(* CoDeSys 2.3 export: PUMP_STATION.EXP *)
(* Libraries: ANALYZATION.LIB 5.10.99 09:05:06, IECSFC.LIB 13.4.06 15:51:28, STANDARD.LIB 4.10.05 11:14:46, SYSLIBCALLBACK.LIB 26.10.21 13:46:42, SYSLIBTIME.LIB 26.10.21 13:46:42, SYSTASKINFO.LIB 26.10.21 13:46:42, Util.lib 18.5.10 15:14:28 *)

(* PLC configuration (modules and I/O channels)
PLC110_32 [Root] node -1, in %IB0 out %QB0 {param 1 = PLC110-32_v2; param 2 = 1; param 3 = 1000}
  Fast discrete inputs [I_SIMPLE_INPUT] node 0, in %IB0 out %QB0 {param 1 = Fast discrete inputs; param 2 = 10000}
    AT %IX0.0 [BitInput] Discrete input 1 {param 1 = Enter name}
    AT %IX0.1 [BitInput] Discrete input 2 {param 1 = Enter name}
  Discrete inputs [ID130] node 1, in %IB1 out %QB1 {param 1 = Discrete inputs; param 2 = 16; param 3 = 16}
    discrete_input_first_byte AT %IB1.0 [ByteInput] discrete_input_first_byte {param 1 = Enter name}
    discrete_input_second_byte AT %IB1.1 [ByteInput] discrete input_second_byte {param 1 = Enter name}
  Fast discrete outputs [OWEN_ID570] node 2, in %IB2 out %QB2 {param 1 = Fast discrete outputs; param 2 = FALSE; param 3 = FALSE; param 4 = FALSE; param 5 = FALSE}
    hw_run_id1 AT %QX2.0 [BitOutput] Run hot water invertor drive1 {param 1 = Enter name}
    hw_run_id2 AT %QX2.1 [BitOutput] Run hot water invertor drive2 {param 1 = Enter name}
    ws_run_id1 AT %QX2.2 [BitOutput] Run water supply invertor drive1 {param 1 = Enter name}
    ws_run_id2 AT %QX2.3 [BitOutput] Run water supply invertor drive2 {param 1 = Enter name}
  Discrete outputs [ID131] node 3, in %IB3 out %QB3 {param 1 = Discrete outputs; param 2 = 0; param 3 = 0; param 4 = 0; param 5 = 24}
    AT %QB3.0 [ByteOutput] 8 discrete outputs {param 1 = Enter name}
    AT %QB3.1 [ByteOutput] 8 discrete outputs {param 1 = Enter name}
  Special input [ID103] node 4, in %IB4 out %QB4 {param 1 = Special input}
    AT %IX4.0 [BitInput] Special input {param 1 = Enter name}
  Special output [ID104] node 5, in %IB5 out %QB5 {param 1 = Special output}
    AT %QX5.0 [BitOutput] Special output {param 1 = Enter name}
  ModBus (Master) [MODBUS_MASTER_ID450] node 6, in %IB6 out %QB6 {param 1 = ModBus (Master); param 2 = No}
    AT %QD6.0 [DWordOutput] Last address {param 1 = Enter name}
    AT %QW6.1 [WordOutput] Last error {param 1 = Enter name}
    RS-485-1 [COM1_USART] node 0, in %IB6.0 out %QB6.0 {param 1 = RS-485-1; param 2 = 115200; param 3 = NO PARITY CHECK; param 4 = 8 bits; param 5 = One stop bit; param 6 = RS485; param 7 = RTU; param 8 = 0; param 9 = No}
    Universal Modbus device [ID2000] node 1, in %IB6.1 out %QB6.1 {param 1 = Universal Modbus device; param 2 = 10:0:0:223; param 3 = 150; param 4 = 502; param 5 = Serial; param 6 = 16; param 7 = By poll time; param 8 = 100; param 9 = No; param 10 = 0; param 11 = Trace_mode}
      AT %QB6.1.0 [ComChannel] Command (0xff - Start) {param 1 = Enter name}
      Real input module [ID2007] node 0, in %IB6.1.0 out %QB6.1.0 {param 1 = float input module; param 2 = 4; param 3 = Read holding Registers  (0x03); param 8 = No}
        hw_input_pressure AT %QD6.1.0.0 [FloatOutput] {param 1 = Enter name}
      Register input module [ID2003] node 1, in %IB6.1.1 out %QB6.1.1 {param 1 = Register input module; param 2 = 2; param 3 = Read holding Registers  (0x03); param 8 = No}
        hw_error_input_pressure AT %QW6.1.1.0 [WordOutput] {param 1 = Enter name}
      Real input module [ID2007] node 2, in %IB6.1.2 out %QB6.1.2 {param 1 = float input module; param 2 = 10; param 3 = Read holding Registers  (0x03); param 8 = No}
        hw_output_pressure AT %QD6.1.2.0 [FloatOutput] {param 1 = Enter name}
      Register input module [ID2003] node 3, in %IB6.1.3 out %QB6.1.3 {param 1 = Register input module; param 2 = 8; param 3 = Read holding Registers  (0x03); param 8 = No}
        hw_error_output_pressure AT %QW6.1.3.0 [WordOutput] {param 1 = Enter name}
      Real input module [ID2007] node 4, in %IB6.1.4 out %QB6.1.4 {param 1 = float input module; param 2 = 16; param 3 = Read holding Registers  (0x03); param 8 = No}
        ws_input_pressure AT %QD6.1.4.0 [FloatOutput] {param 1 = Enter name}
      Register input module [ID2003] node 5, in %IB6.1.5 out %QB6.1.5 {param 1 = Register input module; param 2 = 14; param 3 = Read holding Registers  (0x03); param 8 = No}
        ws_error_input_pressure AT %QW6.1.5.0 [WordOutput] {param 1 = Enter name}
      Real input module [ID2007] node 6, in %IB6.1.6 out %QB6.1.6 {param 1 = float input module; param 2 = 22; param 3 = Read holding Registers  (0x03); param 8 = No}
        ws_output_pressure AT %QD6.1.6.0 [FloatOutput] {param 1 = Enter name}
      Register input module [ID2003] node 7, in %IB6.1.7 out %QB6.1.7 {param 1 = Register input module; param 2 = 20; param 3 = Read holding Registers  (0x03); param 8 = No}
        ws_error_output_pressure AT %QW6.1.7.0 [WordOutput] {param 1 = Enter name}
  ModBus (Master) [MODBUS_MASTER_ID450] node 7, in %IB7 out %QB7 {param 1 = ModBus (Master); param 2 = No}
    AT %QD7.0 [DWordOutput] Last address {param 1 = Enter name}
    AT %QW7.1 [WordOutput] Last error {param 1 = Enter name}
    RS-485-1 [COM1_USART] node 0, in %IB7.0 out %QB7.0 {param 1 = RS-485-1; param 2 = 115200; param 3 = NO PARITY CHECK; param 4 = 8 bits; param 5 = One stop bit; param 6 = RS485; param 7 = RTU; param 8 = 0; param 9 = No}
    Universal Modbus device [ID2000] node 1, in %IB7.1 out %QB7.1 {param 1 = Universal Modbus device; param 2 = 10:0:0:223; param 3 = 150; param 4 = 502; param 5 = Serial; param 6 = 32; param 7 = By poll time; param 8 = 100; param 9 = No; param 10 = 0; param 11 = Trace_mode}
      AT %QB7.1.0 [ComChannel] Command (0xff - Start) {param 1 = Enter name}
      Register output module [ID2004] node 0, in %IB7.1.0 out %QB7.1.0 {param 1 = Register; param 2 = 0; param 3 = Write multiple registers(0x10); param 8 = No}
        hw_output_value_id1 AT %QW7.1.0.0 [WordOutput] {param 1 = Enter name}
      Register output module [ID2004] node 1, in %IB7.1.1 out %QB7.1.1 {param 1 = Register; param 2 = 1; param 3 = Write multiple registers(0x10); param 8 = No}
        hw_output_value_id2 AT %QW7.1.1.0 [WordOutput] {param 1 = Enter name}
      Register output module [ID2004] node 2, in %IB7.1.2 out %QB7.1.2 {param 1 = Register; param 2 = 2; param 3 = Write multiple registers(0x10); param 8 = No}
        ws_output_value_id1 AT %QW7.1.2.0 [WordOutput] {param 1 = Enter name}
      Register output module [ID2004] node 3, in %IB7.1.3 out %QB7.1.3 {param 1 = Register; param 2 = 3; param 3 = Write multiple registers(0x10); param 8 = No}
        ws_output_value_id2 AT %QW7.1.3.0 [WordOutput] {param 1 = Enter name}
      Register output module [ID2004] node 4, in %IB7.1.4 out %QB7.1.4 {param 1 = Register; param 2 = 4; param 3 = Write multiple registers(0x10); param 8 = No}
        AT %QW7.1.4.0 [WordOutput] {param 1 = Enter name}
      Register output module [ID2004] node 5, in %IB7.1.5 out %QB7.1.5 {param 1 = Register; param 2 = 5; param 3 = Write multiple registers(0x10); param 8 = No}
        AT %QW7.1.5.0 [WordOutput] {param 1 = Enter name}
      Register output module [ID2004] node 6, in %IB7.1.6 out %QB7.1.6 {param 1 = Register; param 2 = 6; param 3 = Write multiple registers(0x10); param 8 = No}
        AT %QW7.1.6.0 [WordOutput] {param 1 = Enter name}
      Register output module [ID2004] node 7, in %IB7.1.7 out %QB7.1.7 {param 1 = Register; param 2 = 7; param 3 = Write multiple registers(0x10); param 8 = No}
        AT %QW7.1.7.0 [WordOutput] {param 1 = Enter name}
  ModBus (slave) [MODBUS_ID400] node 8, in %IB8 out %QB8 {param 1 = ModBus (slave); param 2 = 1}
    Modbus [MODBUS_ID302] node 0, in %IB8.0 out %QB8.0 {param 1 = Modbus}
      RS-232 [COM2_USART] node 0, in %IB8.0.0 out %QB8.0.0 {param 1 = RS-232; param 2 = 115200; param 3 = NO PARITY CHECK; param 4 = 8 bits; param 5 = One stop bit; param 6 = RS232; param 7 = RTU; param 8 = 0; param 9 = No}
    8 bits [8Bit] node 1, in %IB8.1 out %QB8.1 {param 1 = 8 bit}
      AT %QB8.1.0 [ByteOutput] {param 1 = Enter name}
    8 bits [8Bit] node 2, in %IB8.2 out %QB8.2 {param 1 = 8 bit}
      AT %QB8.2.0 [ByteOutput] {param 1 = Enter name}
    8 bits [8Bit] node 3, in %IB8.3 out %QB8.3 {param 1 = 8 bit}
      AT %QB8.3.0 [ByteOutput] {param 1 = Enter name}
    8 bits [8Bit] node 4, in %IB8.4 out %QB8.4 {param 1 = 8 bit}
      AT %QB8.4.0 [ByteOutput] {param 1 = Enter name}
    2 byte [Register] node 5, in %IB8.5 out %QB8.5 {param 1 = 2 byte}
      hw_pivot_single AT %QW8.5.0 [WordOutput] {param 1 = Enter name}
    2 byte [Register] node 6, in %IB8.6 out %QB8.6 {param 1 = 2 byte}
      hw_pivot_cascade AT %QW8.6.0 [WordOutput] {param 1 = Enter name}
    2 byte [Register] node 7, in %IB8.7 out %QB8.7 {param 1 = 2 byte}
      hw_cycle_set_hours AT %QW8.7.0 [WordOutput] {param 1 = Enter name}
    2 byte [Register] node 8, in %IB8.8 out %QB8.8 {param 1 = 2 byte}
      hw_cycle_set_minutes AT %QW8.8.0 [WordOutput] {param 1 = Enter name}
    2 byte [Register] node 9, in %IB8.9 out %QB8.9 {param 1 = 2 byte}
      hw_cycle_set_seconds AT %QW8.9.0 [WordOutput] {param 1 = Enter name}
    2 byte [Register] node 10, in %IB8.10 out %QB8.10 {param 1 = 2 byte}
      hw_cascade_delay_on_hours AT %QW8.10.0 [WordOutput] {param 1 = Enter name}
    2 byte [Register] node 11, in %IB8.11 out %QB8.11 {param 1 = 2 byte}
      hw_cascade_delay_on_minutes AT %QW8.11.0 [WordOutput] {param 1 = Enter name}
    2 byte [Register] node 12, in %IB8.12 out %QB8.12 {param 1 = 2 byte}
      hw_cascade_delay_on_seconds AT %QW8.12.0 [WordOutput] {param 1 = Enter name}
    2 byte [Register] node 13, in %IB8.13 out %QB8.13 {param 1 = 2 byte}
      hw_cascade_delay_off_hours AT %QW8.13.0 [WordOutput] {param 1 = Enter name}
    2 byte [Register] node 14, in %IB8.14 out %QB8.14 {param 1 = 2 byte}
      hw_cascade_delay_off_minutes AT %QW8.14.0 [WordOutput] {param 1 = Enter name}
    2 byte [Register] node 15, in %IB8.15 out %QB8.15 {param 1 = 2 byte}
      hw_cascade_delay_off_seconds AT %QW8.15.0 [WordOutput] {param 1 = Enter name}
    2 byte [Register] node 16, in %IB8.16 out %QB8.16 {param 1 = 2 byte}
      ws_pivot_single AT %QW8.16.0 [WordOutput] {param 1 = Enter name}
    2 byte [Register] node 17, in %IB8.17 out %QB8.17 {param 1 = 2 byte}
      ws_pivot_cascade AT %QW8.17.0 [WordOutput] {param 1 = Enter name}
    2 byte [Register] node 18, in %IB8.18 out %QB8.18 {param 1 = 2 byte}
      ws_cycle_set_hours AT %QW8.18.0 [WordOutput] {param 1 = Enter name}
    2 byte [Register] node 19, in %IB8.19 out %QB8.19 {param 1 = 2 byte}
      ws_cycle_set_minutes AT %QW8.19.0 [WordOutput] {param 1 = Enter name}
    2 byte [Register] node 20, in %IB8.20 out %QB8.20 {param 1 = 2 byte}
      ws_cycle_set_seconds AT %QW8.20.0 [WordOutput] {param 1 = Enter name}
    2 byte [Register] node 21, in %IB8.21 out %QB8.21 {param 1 = 2 byte}
      ws_cascade_delay_on_hours AT %QW8.21.0 [WordOutput] {param 1 = Enter name}
    2 byte [Register] node 22, in %IB8.22 out %QB8.22 {param 1 = 2 byte}
      ws_cascade_delay_on_minutes AT %QW8.22.0 [WordOutput] {param 1 = Enter name}
    2 byte [Register] node 23, in %IB8.23 out %QB8.23 {param 1 = 2 byte}
      ws_cascade_delay_on_seconds AT %QW8.23.0 [WordOutput] {param 1 = Enter name}
    2 byte [Register] node 24, in %IB8.24 out %QB8.24 {param 1 = 2 byte}
      ws_cascade_delay_off_hours AT %QW8.24.0 [WordOutput] {param 1 = Enter name}
    2 byte [Register] node 25, in %IB8.25 out %QB8.25 {param 1 = 2 byte}
      ws_cascade_delay_off_minutes AT %QW8.25.0 [WordOutput] {param 1 = Enter name}
    2 byte [Register] node 26, in %IB8.26 out %QB8.26 {param 1 = 2 byte}
      ws_cascade_delay_off_seconds AT %QW8.26.0 [WordOutput] {param 1 = Enter name}
    Float [Float] node 27, in %IB8.27 out %QB8.27 {param 1 = float}
      hw_set_point_pressure AT %QD8.27.0 [FloatOutput] {param 1 = Enter name}
    Float [Float] node 28, in %IB8.28 out %QB8.28 {param 1 = float}
      ws_set_point_pressure AT %QD8.28.0 [FloatOutput] {param 1 = Enter name}
    Float [Float] node 29, in %IB8.29 out %QB8.29 {param 1 = float}
      hw_min_measure_range_input AT %QD8.29.0 [FloatOutput] {param 1 = Enter name}
    Float [Float] node 30, in %IB8.30 out %QB8.30 {param 1 = float}
      hw_max_measure_range_input AT %QD8.30.0 [FloatOutput] {param 1 = Enter name}
    Float [Float] node 31, in %IB8.31 out %QB8.31 {param 1 = float}
      hw_min_measure_range_output AT %QD8.31.0 [FloatOutput] {param 1 = Enter name}
    Float [Float] node 32, in %IB8.32 out %QB8.32 {param 1 = float}
      hw_max_measure_range_output AT %QD8.32.0 [FloatOutput] {param 1 = Enter name}
    Float [Float] node 33, in %IB8.33 out %QB8.33 {param 1 = float}
      ws_min_measure_range_input AT %QD8.33.0 [FloatOutput] {param 1 = Enter name}
    Float [Float] node 34, in %IB8.34 out %QB8.34 {param 1 = float}
      ws_max_measure_range_input AT %QD8.34.0 [FloatOutput] {param 1 = Enter name}
    Float [Float] node 35, in %IB8.35 out %QB8.35 {param 1 = float}
      ws_min_measure_range_output AT %QD8.35.0 [FloatOutput] {param 1 = Enter name}
    Float [Float] node 36, in %IB8.36 out %QB8.36 {param 1 = float}
      ws_max_measure_range_output AT %QD8.36.0 [FloatOutput] {param 1 = Enter name}
    Float [Float] node 37, in %IB8.37 out %QB8.37 {param 1 = float}
      hw_input_pressure_bar AT %QD8.37.0 [FloatOutput] {param 1 = Enter name}
    Float [Float] node 38, in %IB8.38 out %QB8.38 {param 1 = float}
      hw_output_pressure_bar AT %QD8.38.0 [FloatOutput] {param 1 = Enter name}
    Float [Float] node 39, in %IB8.39 out %QB8.39 {param 1 = float}
      ws_input_pressure_bar AT %QD8.39.0 [FloatOutput] {param 1 = Enter name}
    Float [Float] node 40, in %IB8.40 out %QB8.40 {param 1 = float}
      ws_output_pressure_bar AT %QD8.40.0 [FloatOutput] {param 1 = Enter name}
    Float [Float] node 41, in %IB8.41 out %QB8.41 {param 1 = float}
      hw_frequency_id1 AT %QD8.41.0 [FloatOutput] {param 1 = Enter name}
    Float [Float] node 42, in %IB8.42 out %QB8.42 {param 1 = float}
      hw_frequency_id2 AT %QD8.42.0 [FloatOutput] {param 1 = Enter name}
    Float [Float] node 43, in %IB8.43 out %QB8.43 {param 1 = float}
      ws_frequency_id1 AT %QD8.43.0 [FloatOutput] {param 1 = Enter name}
    Float [Float] node 44, in %IB8.44 out %QB8.44 {param 1 = float}
      ws_frequency_id2 AT %QD8.44.0 [FloatOutput] {param 1 = Enter name}
    2 byte [Register] node 45, in %IB8.45 out %QB8.45 {param 1 = 2 byte}
      hw_alarm_error_code AT %QW8.45.0 [WordOutput] {param 1 = Enter name}
    2 byte [Register] node 46, in %IB8.46 out %QB8.46 {param 1 = 2 byte}
      ws_alarm_error_code AT %QW8.46.0 [WordOutput] {param 1 = Enter name}
    Float [Float] node 47, in %IB8.47 out %QB8.47 {param 1 = float}
      hw_manual_set_frequency_id1 AT %QD8.47.0 [FloatOutput] {param 1 = Enter name}
    Float [Float] node 48, in %IB8.48 out %QB8.48 {param 1 = float}
      hw_manual_set_frequency_id2 AT %QD8.48.0 [FloatOutput] {param 1 = Enter name}
    Float [Float] node 49, in %IB8.49 out %QB8.49 {param 1 = float}
      ws_manual_set_frequency_id1 AT %QD8.49.0 [FloatOutput] {param 1 = Enter name}
    Float [Float] node 50, in %IB8.50 out %QB8.50 {param 1 = float}
      ws_manual_set_frequency_id2 AT %QD8.50.0 [FloatOutput] {param 1 = Enter name}
    2 byte [Register] node 51, in %IB8.51 out %QB8.51 {param 1 = 2 byte}
      AT %QW8.51.0 [WordOutput] {param 1 = Enter name}
    2 byte [Register] node 52, in %IB8.52 out %QB8.52 {param 1 = 2 byte}
      AT %QW8.52.0 [WordOutput] {param 1 = Enter name}
    2 byte [Register] node 53, in %IB8.53 out %QB8.53 {param 1 = 2 byte}
      AT %QW8.53.0 [WordOutput] {param 1 = Enter name}
    2 byte [Register] node 54, in %IB8.54 out %QB8.54 {param 1 = 2 byte}
      AT %QW8.54.0 [WordOutput] {param 1 = Enter name}
    2 byte [Register] node 55, in %IB8.55 out %QB8.55 {param 1 = 2 byte}
      AT %QW8.55.0 [WordOutput] {param 1 = Enter name}
    2 byte [Register] node 56, in %IB8.56 out %QB8.56 {param 1 = 2 byte}
      AT %QW8.56.0 [WordOutput] {param 1 = Enter name}
    2 byte [Register] node 57, in %IB8.57 out %QB8.57 {param 1 = 2 byte}
      AT %QW8.57.0 [WordOutput] {param 1 = Enter name}
    2 byte [Register] node 58, in %IB8.58 out %QB8.58 {param 1 = 2 byte}
      AT %QW8.58.0 [WordOutput] {param 1 = Enter name}
    2 byte [Register] node 59, in %IB8.59 out %QB8.59 {param 1 = 2 byte}
      AT %QW8.59.0 [WordOutput] {param 1 = Enter name}
    2 byte [Register] node 60, in %IB8.60 out %QB8.60 {param 1 = 2 byte}
      AT %QW8.60.0 [WordOutput] {param 1 = Enter name}
    2 byte [Register] node 61, in %IB8.61 out %QB8.61 {param 1 = 2 byte}
      AT %QW8.61.0 [WordOutput] {param 1 = Enter name}
    2 byte [Register] node 62, in %IB8.62 out %QB8.62 {param 1 = 2 byte}
      AT %QW8.62.0 [WordOutput] {param 1 = Enter name}
    2 byte [Register] node 63, in %IB8.63 out %QB8.63 {param 1 = 2 byte}
      AT %QW8.63.0 [WordOutput] {param 1 = Enter name}
    2 byte [Register] node 64, in %IB8.64 out %QB8.64 {param 1 = 2 byte}
      AT %QW8.64.0 [WordOutput] {param 1 = Enter name}
    2 byte [Register] node 65, in %IB8.65 out %QB8.65 {param 1 = 2 byte}
      AT %QW8.65.0 [WordOutput] {param 1 = Enter name}
    2 byte [Register] node 66, in %IB8.66 out %QB8.66 {param 1 = 2 byte}
      AT %QW8.66.0 [WordOutput] {param 1 = Enter name}
    2 byte [Register] node 67, in %IB8.67 out %QB8.67 {param 1 = 2 byte}
      AT %QW8.67.0 [WordOutput] {param 1 = Enter name}
    2 byte [Register] node 68, in %IB8.68 out %QB8.68 {param 1 = 2 byte}
      AT %QW8.68.0 [WordOutput] {param 1 = Enter name}
    2 byte [Register] node 69, in %IB8.69 out %QB8.69 {param 1 = 2 byte}
      AT %QW8.69.0 [WordOutput] {param 1 = Enter name}
    2 byte [Register] node 70, in %IB8.70 out %QB8.70 {param 1 = 2 byte}
      AT %QW8.70.0 [WordOutput] {param 1 = Enter name}
    2 byte [Register] node 71, in %IB8.71 out %QB8.71 {param 1 = 2 byte}
      AT %QW8.71.0 [WordOutput] {param 1 = Enter name}
    2 byte [Register] node 72, in %IB8.72 out %QB8.72 {param 1 = 2 byte}
      AT %QW8.72.0 [WordOutput] {param 1 = Enter name}
    2 byte [Register] node 73, in %IB8.73 out %QB8.73 {param 1 = 2 byte}
      AT %QW8.73.0 [WordOutput] {param 1 = Enter name}
    2 byte [Register] node 74, in %IB8.74 out %QB8.74 {param 1 = 2 byte}
      AT %QW8.74.0 [WordOutput] {param 1 = Enter name}
    2 byte [Register] node 75, in %IB8.75 out %QB8.75 {param 1 = 2 byte}
      AT %QW8.75.0 [WordOutput] {param 1 = Enter name}
    2 byte [Register] node 76, in %IB8.76 out %QB8.76 {param 1 = 2 byte}
      AT %QW8.76.0 [WordOutput] {param 1 = Enter name}
    2 byte [Register] node 77, in %IB8.77 out %QB8.77 {param 1 = 2 byte}
      AT %QW8.77.0 [WordOutput] {param 1 = Enter name}
    2 byte [Register] node 78, in %IB8.78 out %QB8.78 {param 1 = 2 byte}
      AT %QW8.78.0 [WordOutput] {param 1 = Enter name}
    2 byte [Register] node 79, in %IB8.79 out %QB8.79 {param 1 = 2 byte}
      AT %QW8.79.0 [WordOutput] {param 1 = Enter name}
    2 byte [Register] node 80, in %IB8.80 out %QB8.80 {param 1 = 2 byte}
      AT %QW8.80.0 [WordOutput] {param 1 = Enter name}
    2 byte [Register] node 81, in %IB8.81 out %QB8.81 {param 1 = 2 byte}
      AT %QW8.81.0 [WordOutput] {param 1 = Enter name}
    2 byte [Register] node 82, in %IB8.82 out %QB8.82 {param 1 = 2 byte}
      AT %QW8.82.0 [WordOutput] {param 1 = Enter name}
    2 byte [Register] node 83, in %IB8.83 out %QB8.83 {param 1 = 2 byte}
      AT %QW8.83.0 [WordOutput] {param 1 = Enter name}
    2 byte [Register] node 84, in %IB8.84 out %QB8.84 {param 1 = 2 byte}
      AT %QW8.84.0 [WordOutput] {param 1 = Enter name}
    2 byte [Register] node 85, in %IB8.85 out %QB8.85 {param 1 = 2 byte}
      AT %QW8.85.0 [WordOutput] {param 1 = Enter name}
    2 byte [Register] node 86, in %IB8.86 out %QB8.86 {param 1 = 2 byte}
      AT %QW8.86.0 [WordOutput] {param 1 = Enter name}
    2 byte [Register] node 87, in %IB8.87 out %QB8.87 {param 1 = 2 byte}
      AT %QW8.87.0 [WordOutput] {param 1 = Enter name}
    2 byte [Register] node 88, in %IB8.88 out %QB8.88 {param 1 = 2 byte}
      AT %QW8.88.0 [WordOutput] {param 1 = Enter name}
    2 byte [Register] node 89, in %IB8.89 out %QB8.89 {param 1 = 2 byte}
      AT %QW8.89.0 [WordOutput] {param 1 = Enter name}
    2 byte [Register] node 90, in %IB8.90 out %QB8.90 {param 1 = 2 byte}
      AT %QW8.90.0 [WordOutput] {param 1 = Enter name}
    2 byte [Register] node 91, in %IB8.91 out %QB8.91 {param 1 = 2 byte}
      AT %QW8.91.0 [WordOutput] {param 1 = Enter name}
    2 byte [Register] node 92, in %IB8.92 out %QB8.92 {param 1 = 2 byte}
      AT %QW8.92.0 [WordOutput] {param 1 = Enter name}
    2 byte [Register] node 93, in %IB8.93 out %QB8.93 {param 1 = 2 byte}
      AT %QW8.93.0 [WordOutput] {param 1 = Enter name}
    2 byte [Register] node 94, in %IB8.94 out %QB8.94 {param 1 = 2 byte}
      AT %QW8.94.0 [WordOutput] {param 1 = Enter name}
    2 byte [Register] node 95, in %IB8.95 out %QB8.95 {param 1 = 2 byte}
      AT %QW8.95.0 [WordOutput] {param 1 = Enter name}
    2 byte [Register] node 96, in %IB8.96 out %QB8.96 {param 1 = 2 byte}
      AT %QW8.96.0 [WordOutput] {param 1 = Enter name}
    2 byte [Register] node 97, in %IB8.97 out %QB8.97 {param 1 = 2 byte}
      AT %QW8.97.0 [WordOutput] {param 1 = Enter name}
    2 byte [Register] node 98, in %IB8.98 out %QB8.98 {param 1 = 2 byte}
      AT %QW8.98.0 [WordOutput] {param 1 = Enter name}
    2 byte [Register] node 99, in %IB8.99 out %QB8.99 {param 1 = 2 byte}
      AT %QW8.99.0 [WordOutput] {param 1 = Enter name}
    2 byte [Register] node 100, in %IB8.100 out %QB8.100 {param 1 = 2 byte}
      AT %QW8.100.0 [WordOutput] {param 1 = Enter name}
    2 byte [Register] node 101, in %IB8.101 out %QB8.101 {param 1 = 2 byte}
      AT %QW8.101.0 [WordOutput] {param 1 = Enter name}
    2 byte [Register] node 102, in %IB8.102 out %QB8.102 {param 1 = 2 byte}
      AT %QW8.102.0 [WordOutput] {param 1 = Enter name}
    2 byte [Register] node 103, in %IB8.103 out %QB8.103 {param 1 = 2 byte}
      AT %QW8.103.0 [WordOutput] {param 1 = Enter name}
    2 byte [Register] node 104, in %IB8.104 out %QB8.104 {param 1 = 2 byte}
      AT %QW8.104.0 [WordOutput] {param 1 = Enter name}
    2 byte [Register] node 105, in %IB8.105 out %QB8.105 {param 1 = 2 byte}
      AT %QW8.105.0 [WordOutput] {param 1 = Enter name}
    2 byte [Register] node 106, in %IB8.106 out %QB8.106 {param 1 = 2 byte}
      AT %QW8.106.0 [WordOutput] {param 1 = Enter name}
    2 byte [Register] node 107, in %IB8.107 out %QB8.107 {param 1 = 2 byte}
      AT %QW8.107.0 [WordOutput] {param 1 = Enter name}
    2 byte [Register] node 108, in %IB8.108 out %QB8.108 {param 1 = 2 byte}
      AT %QW8.108.0 [WordOutput] {param 1 = Enter name}
    2 byte [Register] node 109, in %IB8.109 out %QB8.109 {param 1 = 2 byte}
      AT %QW8.109.0 [WordOutput] {param 1 = Enter name}
    2 byte [Register] node 110, in %IB8.110 out %QB8.110 {param 1 = 2 byte}
      AT %QW8.110.0 [WordOutput] {param 1 = Enter name}
    2 byte [Register] node 111, in %IB8.111 out %QB8.111 {param 1 = 2 byte}
      AT %QW8.111.0 [WordOutput] {param 1 = Enter name}
    2 byte [Register] node 112, in %IB8.112 out %QB8.112 {param 1 = 2 byte}
      AT %QW8.112.0 [WordOutput] {param 1 = Enter name}
    2 byte [Register] node 113, in %IB8.113 out %QB8.113 {param 1 = 2 byte}
      AT %QW8.113.0 [WordOutput] {param 1 = Enter name}
    2 byte [Register] node 114, in %IB8.114 out %QB8.114 {param 1 = 2 byte}
      AT %QW8.114.0 [WordOutput] {param 1 = Enter name}
    2 byte [Register] node 115, in %IB8.115 out %QB8.115 {param 1 = 2 byte}
      AT %QW8.115.0 [WordOutput] {param 1 = Enter name}
    2 byte [Register] node 116, in %IB8.116 out %QB8.116 {param 1 = 2 byte}
      AT %QW8.116.0 [WordOutput] {param 1 = Enter name}
    2 byte [Register] node 117, in %IB8.117 out %QB8.117 {param 1 = 2 byte}
      AT %QW8.117.0 [WordOutput] {param 1 = Enter name}
    2 byte [Register] node 118, in %IB8.118 out %QB8.118 {param 1 = 2 byte}
      AT %QW8.118.0 [WordOutput] {param 1 = Enter name}
    2 byte [Register] node 119, in %IB8.119 out %QB8.119 {param 1 = 2 byte}
      AT %QW8.119.0 [WordOutput] {param 1 = Enter name}
    2 byte [Register] node 120, in %IB8.120 out %QB8.120 {param 1 = 2 byte}
      AT %QW8.120.0 [WordOutput] {param 1 = Enter name}
    2 byte [Register] node 121, in %IB8.121 out %QB8.121 {param 1 = 2 byte}
      AT %QW8.121.0 [WordOutput] {param 1 = Enter name}
    2 byte [Register] node 122, in %IB8.122 out %QB8.122 {param 1 = 2 byte}
      AT %QW8.122.0 [WordOutput] {param 1 = Enter name}
    2 byte [Register] node 123, in %IB8.123 out %QB8.123 {param 1 = 2 byte}
      AT %QW8.123.0 [WordOutput] {param 1 = Enter name}
    2 byte [Register] node 124, in %IB8.124 out %QB8.124 {param 1 = 2 byte}
      AT %QW8.124.0 [WordOutput] {param 1 = Enter name}
    2 byte [Register] node 125, in %IB8.125 out %QB8.125 {param 1 = 2 byte}
      AT %QW8.125.0 [WordOutput] {param 1 = Enter name}
    2 byte [Register] node 126, in %IB8.126 out %QB8.126 {param 1 = 2 byte}
      AT %QW8.126.0 [WordOutput] {param 1 = Enter name}
    2 byte [Register] node 127, in %IB8.127 out %QB8.127 {param 1 = 2 byte}
      AT %QW8.127.0 [WordOutput] {param 1 = Enter name}
    2 byte [Register] node 128, in %IB8.128 out %QB8.128 {param 1 = 2 byte}
      AT %QW8.128.0 [WordOutput] {param 1 = Enter name}
    2 byte [Register] node 129, in %IB8.129 out %QB8.129 {param 1 = 2 byte}
      AT %QW8.129.0 [WordOutput] {param 1 = Enter name}
    2 byte [Register] node 130, in %IB8.130 out %QB8.130 {param 1 = 2 byte}
      AT %QW8.130.0 [WordOutput] {param 1 = Enter name}
    2 byte [Register] node 131, in %IB8.131 out %QB8.131 {param 1 = 2 byte}
      AT %QW8.131.0 [WordOutput] {param 1 = Enter name}
*)

(* Data type in CascadeMode *)
TYPE classInfoCascade :

STRUCT
	pivot:INT;
	error_message:STRING(79);
	error_code: WORD;
	cascade_pump1:classInfoCascadePump;
	cascade_pump2:classInfoCascadePump;
	cascade_pump3:classInfoCascadePump;
	cascade_pump4:classInfoCascadePump;
	cascade_pump5:classInfoCascadePump;
	cascade_pump6:classInfoCascadePump;
	cascade_pump7:classInfoCascadePump;
	cascade_pump8:classInfoCascadePump;
END_STRUCT

END_TYPE

(* Data type in CascadeMode *)
TYPE classInfoCascadePump :

STRUCT
	cascade_pump:BOOL := FALSE;  (*ï¿½ï¿½ï¿½ï¿½ï¿½ï¿½ ï¿½ï¿½ï¿½ï¿½ï¿½ï¿½ ï¿½ï¿½ï¿½ï¿½ï¿½ï¿½*)
	manual:INT := 40;  (*Hz*)
END_STRUCT

END_TYPE

(* Data type in CycleMode *)
TYPE classInfoCycle :

STRUCT
	run_timer: BOOL; (* status work *)
	working_time: TIME; (* pump working time  *)
	pump_number: INT;  (* number working pump *)
	error_code:  WORD;
END_STRUCT

END_TYPE

(* Data type in InvertorDrive/set_auto_invertor_drive *)
TYPE classSetAutoInvertorDrive :

STRUCT
	auto:BOOL := FALSE;
	direct_logic:BOOL := TRUE;  (* ï¿½ï¿½ï¿½ï¿½ ï¿½ï¿½ï¿½ï¿½ï¿½ï¿½ï¿½/ï¿½ï¿½ï¿½ï¿½ï¿½ï¿½ï¿½ï¿½ï¿½ ï¿½ï¿½ï¿½ï¿½ï¿½ï¿½ï¿½ï¿½ï¿½ï¿½; ï¿½ï¿½ï¿½ ï¿½ï¿½ï¿½ï¿½ï¿½ï¿½ï¿½ï¿½ ï¿½ï¿½ï¿½ï¿½ï¿½ï¿½ï¿½ï¿½ï¿½ï¿½ ï¿½ï¿½ï¿½ï¿½ ï¿½ï¿½ï¿½ï¿½ï¿½ï¿½ï¿½ï¿½ ï¿½ï¿½ï¿½ï¿½ï¿½ï¿½ï¿½ï¿½ï¿½ï¿½ï¿½ï¿½ï¿½ï¿½ ï¿½ï¿½ï¿½ï¿½ï¿½ï¿½ï¿½ï¿½ ï¿½ï¿½ï¿½ï¿½ ï¿½ï¿½ï¿½ï¿½ï¿½ï¿½ï¿½, ï¿½ï¿½ï¿½ï¿½ï¿½ï¿½ï¿½ï¿½ ï¿½ï¿½ï¿½ï¿½ï¿½ï¿½ï¿½ ï¿½ï¿½ï¿½ï¿½ï¿½ï¿½ï¿½ï¿½ï¿½ï¿½ï¿½, ï¿½ ï¿½ï¿½ï¿½ï¿½ï¿½ï¿½ï¿½ï¿½*)
	set_point:REAL := 0;  (* ï¿½ï¿½ï¿½ï¿½ï¿½ï¿½ï¿½, ï¿½ï¿½ï¿½ï¿½ï¿½ï¿½ï¿½ï¿½ ï¿½ ï¿½ï¿½ï¿½ï¿½ï¿½ï¿½ï¿½ï¿½ ï¿½ï¿½ï¿½ï¿½ï¿½ï¿½ï¿½ï¿½ï¿½ ï¿½ï¿½ï¿½ï¿½ï¿½ï¿½ï¿½ï¿½ï¿½ï¿½ï¿½ï¿½ï¿½ï¿½ ï¿½ï¿½ï¿½ï¿½ï¿½ï¿½ï¿½ï¿½ *)
	value:REAL := 0;  (* ï¿½ï¿½ï¿½ï¿½ï¿½ï¿½ï¿½ ï¿½ï¿½ï¿½ï¿½ï¿½ï¿½ï¿½ï¿½ ï¿½ï¿½ï¿½ï¿½ï¿½ï¿½ï¿½ï¿½ï¿½ï¿½ï¿½ï¿½ï¿½ï¿½ ï¿½ï¿½ï¿½ï¿½ï¿½ï¿½ï¿½ï¿½, ï¿½ï¿½ï¿½ï¿½ï¿½ï¿½ï¿½ï¿½ï¿½ï¿½ ï¿½ ï¿½ï¿½ï¿½ï¿½ï¿½ï¿½ï¿½ *)
	P:REAL := 2;  (* ï¿½ï¿½ï¿½ï¿½ï¿½ï¿½ï¿½ï¿½ï¿½ï¿½ï¿½ï¿½ï¿½ï¿½ï¿½ï¿½ ï¿½ï¿½ï¿½ï¿½ï¿½ï¿½ï¿½ï¿½ï¿½ï¿½ï¿½ ï¿½ï¿½ï¿½ï¿½ï¿½ï¿½ï¿½ï¿½ï¿½ï¿½, ï¿½ï¿½ï¿½ ï¿½ï¿½ï¿½ï¿½ï¿½ï¿½ï¿½ï¿½ï¿½ï¿½ ï¿½ï¿½ï¿½ï¿½ï¿½ ï¿½ï¿½ï¿½ï¿½ï¿½ï¿½ï¿½ï¿½ï¿½ï¿½ ï¿½ï¿½ï¿½ï¿½ï¿½ï¿½ï¿½ï¿½ï¿½ï¿½ ï¿½ï¿½ï¿½ï¿½ï¿½ï¿½ï¿½*)
	I:INT := 10;  (* ï¿½ï¿½ï¿½ï¿½ï¿½ï¿½ï¿½ï¿½ï¿½ï¿½ï¿½ï¿½ ï¿½ï¿½ï¿½ï¿½ï¿½ï¿½ï¿½ï¿½ï¿½ï¿½ï¿½ ï¿½ï¿½ï¿½ï¿½ï¿½ï¿½ï¿½ï¿½ï¿½ï¿½, ï¿½ï¿½ï¿½ï¿½ï¿½ ï¿½ ï¿½ï¿½ï¿½ï¿½ï¿½ï¿½ï¿½ï¿½ *)
	D:INT := 0;  (* ï¿½ï¿½ï¿½ï¿½ï¿½ï¿½ï¿½ï¿½ï¿½ï¿½ï¿½ï¿½ï¿½ï¿½ï¿½ï¿½ ï¿½ï¿½ï¿½ï¿½ï¿½ï¿½ï¿½ï¿½ï¿½ï¿½ï¿½ ï¿½ï¿½ï¿½ï¿½ï¿½ï¿½ï¿½ï¿½ï¿½ï¿½, ï¿½ï¿½ï¿½ï¿½ï¿½ ï¿½ ï¿½ï¿½ï¿½ï¿½ï¿½ï¿½ï¿½ï¿½ *)
END_STRUCT

END_TYPE

(* Data type in InvertorDrive/set_limit_frequency *)
TYPE classSetLimitFrequency :

STRUCT
	manual:REAL;  (* Hz *)
	min_range:REAL;  (* Hz *)
	max_range:REAL;  (* Hz *)
END_STRUCT

END_TYPE

(* Data type in InvertorDrive *)
TYPE classAlarmInvertorDrive :

STRUCT
	external_alarm:STRING(79);
	fault_invertor_drive:STRING(79);
END_STRUCT

END_TYPE

(* Data type in InvertorDrive *)
TYPE classInfoInvertorDrive :

STRUCT
	active:BOOL;
	status_run:STRING(79);
	set_pid:classSetPid;
	alarm:classAlarmInvertorDrive;
	frequency:REAL;  (* Hz *)
	aout_frequency:REAL;  (* mA *)
	run:BOOL;
	reset_fault:BOOL;
END_STRUCT

END_TYPE

(* Data type in InvertorDrive *)
TYPE classInvertorDrive :

STRUCT
	discrete_inputs:classInvertorDriveDiscreteInputs;
	discrete_outputs:classInvertorDriveDiscreteOutputs;
	analog_input:classInvertorDriveAnalogInputs;
	analog_output:classInvertorDriveAnalogOutputs;
	set:classSetInvertorDrive;
	min_frequency:INT;
	max_frequency:INT;
	set_frequency:REAL;
	real_frequency:REAL;(* ï¿½ï¿½ï¿½ï¿½ï¿½ï¿½ï¿½ï¿½ ï¿½ ï¿½ï¿½ï¿½ï¿½ï¿½ï¿½ï¿½ï¿½ï¿½ï¿½ï¿½ ï¿½ï¿½ï¿½ï¿½ï¿½ï¿½ ï¿½ï¿½ï¿½ï¿½ï¿½ï¿½ï¿½ï¿½ï¿½ï¿½ *)
END_STRUCT

END_TYPE

(* Data type in InvertorDrive *)
TYPE classInvertorDriveAnalogInputs :

STRUCT
	set_frequency:REAL;
END_STRUCT

END_TYPE

(* Data type in InvertorDrive *)
TYPE classInvertorDriveAnalogOutputs :

STRUCT
	out_frequency:REAL;
END_STRUCT

END_TYPE

(* Data type in InvertorDrive *)
TYPE classInvertorDriveDiscreteInputs :

STRUCT
	start:BOOL;
	reset_fault:BOOL;
(* external alarm *)
	low_pressure_in:BOOL;
	high_pressure_out:BOOL;
END_STRUCT

END_TYPE

(* Data type in InvertorDrive *)
TYPE classInvertorDriveDiscreteOutputs :

STRUCT
	status_run:BOOL;
	status_alarm:BOOL;
END_STRUCT

END_TYPE

(* Data type in InvertorDrive *)
TYPE classSetInvertorDrive :

STRUCT
	set_auto:classSetAutoInvertorDrive;
	set_frequency:classSetLimitFrequency;
END_STRUCT

END_TYPE

(* Data type in MB110_8A *)
TYPE classInfoAnalogInputChannel :

STRUCT
	current_value:REAL;
	error_message:STRING(79);
END_STRUCT

END_TYPE

(* Data type in MB110_8A *)
TYPE classInfoAnalogInputModule :

STRUCT
	channel1:classInfoAnalogInputChannel;
	channel2:classInfoAnalogInputChannel;
	channel3:classInfoAnalogInputChannel;
	channel4:classInfoAnalogInputChannel;
	channel5:classInfoAnalogInputChannel;
	channel6:classInfoAnalogInputChannel;
	channel7:classInfoAnalogInputChannel;
	channel8:classInfoAnalogInputChannel;
END_STRUCT

END_TYPE

(* Data type in MB110_8A *)
TYPE classSetAnalogInputChannel :

STRUCT
	(* ï¿½ï¿½ï¿½ï¿½ï¿½ï¿½ï¿½ï¿½ï¿½ï¿½ï¿½ï¿½ï¿½ï¿½ï¿½ï¿½ ï¿½ï¿½ï¿½ï¿½ï¿½ï¿½ï¿½ï¿½ï¿½ ï¿½ï¿½ï¿½ï¿½ï¿½ï¿½ ï¿½ï¿½ï¿½ï¿½ï¿½ï¿½. ï¿½ï¿½. ï¿½ï¿½ï¿½ï¿½ï¿½ï¿½ï¿½ï¿½ï¿½ï¿½ ï¿½ï¿½ï¿½ï¿½ï¿½ï¿½ï¿½: ï¿½ï¿½ï¿½ï¿½ï¿½ï¿½ï¿½ï¿½ï¿½ï¿½. ï¿½ï¿½ï¿½ï¿½ï¿½ï¿½ï¿½ ï¿½.2 *)
	(* ï¿½ï¿½ï¿½ï¿½ï¿½ï¿½ï¿½ ï¿½ï¿½ï¿½ ï¿½ ï¿½ï¿½ï¿½ï¿½ï¿½ï¿½ï¿½ï¿½ ï¿½ï¿½ ï¿½ï¿½ï¿½ï¿½ï¿½ï¿½ï¿½ï¿½ï¿½: ï¿½ï¿½ï¿½ ï¿½ï¿½ï¿½ï¿½ï¿½ï¿½ï¿½ 4-20mA  *)
	ain_l: REAL := 0;  (* ï¿½ï¿½ï¿½ï¿½ï¿½ï¿½ï¿½ï¿½ Ain.L *)
	ain_h: REAL := 1000;  (* ï¿½ï¿½ï¿½ï¿½ï¿½ï¿½ï¿½ï¿½ Ain.H *)
	analog_min_value: REAL := 4;  (* ï¿½ï¿½ï¿½ï¿½ï¿½ï¿½ï¿½ï¿½ ï¿½ï¿½ï¿½ï¿½ï¿½ï¿½ ï¿½ï¿½ï¿½ï¿½ï¿½ï¿½ï¿½ ï¿½ï¿½ï¿½ï¿½ï¿½ï¿½ï¿½ ï¿½ï¿½ï¿½ï¿½ï¿½ï¿½ï¿½ï¿½ *)
	analog_max_value: REAL := 20;  (* ï¿½ï¿½ï¿½ï¿½ï¿½ï¿½ï¿½ï¿½ ï¿½ï¿½ï¿½ï¿½ï¿½ï¿½ï¿½ ï¿½ï¿½ï¿½ï¿½ï¿½ï¿½ï¿½ ï¿½ï¿½ï¿½ï¿½ï¿½ï¿½ï¿½ ï¿½ï¿½ï¿½ï¿½ï¿½ï¿½ï¿½ï¿½ *)
END_STRUCT

END_TYPE

(* Data type in MB110_8A *)
TYPE classSetAnalogInputsModule :

STRUCT
	ch1_set:classSetAnalogInputChannel;
	ch2_set:classSetAnalogInputChannel;
	ch3_set:classSetAnalogInputChannel;
	ch4_set:classSetAnalogInputChannel;
	ch5_set:classSetAnalogInputChannel;
	ch6_set:classSetAnalogInputChannel;
	ch7_set:classSetAnalogInputChannel;
	ch8_set:classSetAnalogInputChannel;
END_STRUCT

END_TYPE

(* Data type in MB110_8U *)
TYPE classAnalogOutputChannel :

STRUCT
	current_value: REAL;
END_STRUCT

END_TYPE

(* Data type in MB110_8U *)
TYPE classAnalogOutputModule :

STRUCT
	channel1:classAnalogOutputChannel;
	channel2:classAnalogOutputChannel;
	channel3:classAnalogOutputChannel;
	channel4:classAnalogOutputChannel;
	channel5:classAnalogOutputChannel;
	channel6:classAnalogOutputChannel;
	channel7:classAnalogOutputChannel;
	channel8:classAnalogOutputChannel;
END_STRUCT

END_TYPE

(* Data type in PID_regulator *)
TYPE classSetPid :

STRUCT
	actual:REAL;
	set_point:REAL;
	P:REAL;  (* ï¿½ï¿½ï¿½ï¿½ï¿½ï¿½ï¿½ï¿½ï¿½ï¿½ï¿½ï¿½ï¿½ï¿½ï¿½ï¿½ ï¿½ï¿½ï¿½ï¿½ï¿½ï¿½ï¿½ï¿½ï¿½ï¿½ï¿½ ï¿½ï¿½ï¿½ï¿½ï¿½ï¿½ï¿½ï¿½ï¿½ï¿½, ï¿½ï¿½ï¿½ ï¿½ï¿½ï¿½ï¿½ï¿½ï¿½ï¿½ï¿½ï¿½ï¿½ ï¿½ï¿½ï¿½ï¿½ï¿½ ï¿½ï¿½ï¿½ï¿½ï¿½ï¿½ï¿½ï¿½ï¿½ï¿½ ï¿½ï¿½ï¿½ï¿½ï¿½ï¿½ï¿½ï¿½ï¿½ï¿½ ï¿½ï¿½ï¿½ï¿½ï¿½ï¿½ï¿½*)
	I:INT;  (* ï¿½ï¿½ï¿½ï¿½ï¿½ï¿½ï¿½ï¿½ï¿½ï¿½ï¿½ï¿½ ï¿½ï¿½ï¿½ï¿½ï¿½ï¿½ï¿½ï¿½ï¿½ï¿½ï¿½ ï¿½ï¿½ï¿½ï¿½ï¿½ï¿½ï¿½ï¿½ï¿½ï¿½, ï¿½ï¿½ï¿½ï¿½ï¿½ ï¿½ ï¿½ï¿½ï¿½ï¿½ï¿½ï¿½ï¿½ï¿½ *)
	D:INT;  (* ï¿½ï¿½ï¿½ï¿½ï¿½ï¿½ï¿½ï¿½ï¿½ï¿½ï¿½ï¿½ï¿½ï¿½ï¿½ï¿½ ï¿½ï¿½ï¿½ï¿½ï¿½ï¿½ï¿½ï¿½ï¿½ï¿½ï¿½ ï¿½ï¿½ï¿½ï¿½ï¿½ï¿½ï¿½ï¿½ï¿½ï¿½, ï¿½ï¿½ï¿½ï¿½ï¿½ ï¿½ ï¿½ï¿½ï¿½ï¿½ï¿½ï¿½ï¿½ï¿½ *)
	Y_manual:REAL := 0;
	Y_offset:REAL;
	Y_min:REAL;
	Y_max:REAL;
	manual:BOOL;
	reset:BOOL;
END_STRUCT

END_TYPE

(* Data type in PLC110/DiscreteInputs *)
TYPE classDiscreteInputByte :

STRUCT
	Bit1:BOOL;
	Bit2:BOOL;
	Bit3:BOOL;
	Bit4:BOOL;
	Bit5:BOOL;
	Bit6:BOOL;
	Bit7:BOOL;
	Bit8:BOOL;
END_STRUCT

END_TYPE

(* Data type in PLC110/DiscreteInputs *)
TYPE classDiscreteInputs :

STRUCT
	first_byte:classDiscreteInputByte;
	second_byte:classDiscreteInputByte;
END_STRUCT

END_TYPE

(* Data type in PLC110/DiscreteInputs *)
TYPE classFastDiscreteInputs :

STRUCT
	Bit1:BOOL;
	Bit2:BOOL;
END_STRUCT

END_TYPE

(* Data type in PLC110/DiscreteInputs *)
TYPE classSpecialInput :

STRUCT
	Bit1:BOOL;
END_STRUCT

END_TYPE

(* Data type in PLC110/DiscreteOutputs *)
TYPE classDiscreteOutputByte :

STRUCT
	Bit1:BOOL;
	Bit2:BOOL;
	Bit3:BOOL;
	Bit4:BOOL;
	Bit5:BOOL;
	Bit6:BOOL;
	Bit7:BOOL;
	Bit8:BOOL;
END_STRUCT

END_TYPE

(* Data type in PLC110/DiscreteOutputs *)
TYPE classDiscreteOutputs :

STRUCT
	first_byte:classDiscreteOutputByte;
	second_byte:classDiscreteOutputByte;
END_STRUCT

END_TYPE

(* Data type in PLC110/DiscreteOutputs *)
TYPE classFastDiscreteOutputs :

STRUCT
	Bit1:BOOL;
	Bit2:BOOL;
	Bit3:BOOL;
	Bit4:BOOL;
END_STRUCT

END_TYPE

(* Data type in PLC110/DiscreteOutputs *)
TYPE classSpecialOutput :

STRUCT
	Bit1:BOOL;
END_STRUCT

END_TYPE

(* Data type in PLC110 *)
TYPE classPLC110_32 :

STRUCT
	fast_discrete_inputs:classFastDiscreteInputs;
	discrete_inputs:classDiscreteInputs;
	special_input:classSpecialInput;
	fast_discrete_outputs:classFastDiscreteOutputs;
	discrete_output:classDiscreteOutputs;
	special_output:classSpecialOutput;
END_STRUCT

END_TYPE

(* Data type in PLC110 *)
TYPE classPLC32m2StatusInputs :

STRUCT
	fast_inputs:classFastDiscreteInputs;
	discrete_inputs:classDiscreteInputs;
	special_input:classSpecialInput;
END_STRUCT

END_TYPE

(* Data type in PLC110 *)
TYPE classPLC32m2StatusOutputs :

STRUCT
	fast_outputs:classFastDiscreteOutputs;
	discrete_outputs:classDiscreteOutputs;
	special_output:classSpecialOutput;
END_STRUCT

END_TYPE

(* Data type in PressureSensor_4_20ma *)
TYPE classSetPressureSensor4_20 :

STRUCT
	min_measure_range:REAL:=0;
	max_measure_range:REAL:=16;
	min_current_range:REAL:=4;
	max_current_range:REAL:=20;
END_STRUCT

END_TYPE

(* Data type in SingleMode *)
TYPE classInfoSingle :
(* class for information single mode. *)

STRUCT
    pivot_pump : INT;
    start_pump : BOOL;
    message: STRING(79);
    error_code: WORD;
END_STRUCT

END_TYPE

(* Data type in value_scale *)
TYPE classParamsValueScaling :

STRUCT
	in_min: REAL := 0;
	in_max: REAL := 100;
	out_min: REAL := 0;
	out_max: REAL := 100;

END_STRUCT

END_TYPE

(* POU PLC_PRG, CFC *)
PROGRAM PLC_PRG
VAR
	PLC: PLC110_32m2;
	analog_inputs_module: MB110_8a;
	currents_value_pack: get_info_analog_outputs_module;
	analog_outputs_module: MY110_8u;
	settings_channel_analog_inputs_module: SetChannelsAnalogInputsModule;
	hw_input: CurrentSensorPressure_4_20;
	hw_output: CurrentSensorPressure_4_20;
	ws_input: CurrentSensorPressure_4_20;
	ws_output: CurrentSensorPressure_4_20;
	(*hw_settings_pressure_input: SetCurrentSensorPressure_4_20;
	hw_settings_pressure_output: SetCurrentSensorPressure_4_20;
	ws_settings_pressure_input: SetCurrentSensorPressure_4_20;
	ws_settings_pressure_output: SetCurrentSensorPressure_4_20;*)
	hw_invertor_drive_1: InvertorDrive;
	hw_invertor_drive_2: InvertorDrive;
	ws_invertor_drive_1: InvertorDrive;
	ws_invertor_drive_2: InvertorDrive;
	hw_settings_pid_id_1: params_in_set_PID;
	hw_settings_pid_id_2: params_in_set_PID;
	ws_settings_pid_id_1: params_in_set_PID;
	ws_settings_pid_id_2: params_in_set_PID;
	pid1: PID;
	pid2: PID;
	pid3: PID;
	pid4: PID;
	 hw_frequency_id_1: REAL;
	hw_frequency_id_2: REAL;
	ws_frequency_id_1: REAL;
	ws_frequency_id_2: REAL;
	(* hw_input_pressure_bar: REAL;
	hw_output_pressure_bar: REAL;
	ws_input_pressure_bar: REAL;
	ws_output_pressure_bar: REAL; *)
	hw_single_mode: Single;
	hw_cycle_mode: cycle;
	hw_cascade_mode: cascade;
	hw_mode_selector: Cascade_Cycle_Selector;
	hw_start_id_1: BOOL;
	hw_start_id_2: BOOL;
	info_analog_inputs_module: classInfoAnalogInputModule;
	hw_info_id_1: classInfoInvertorDrive;
	hw_info_id_2: classInfoInvertorDrive;
	ws_info_id_1: classInfoInvertorDrive;
	ws_info_id_2: classInfoInvertorDrive;
	hw_kpi_35: Kpi;
	hw_kpi_36: Kpi;
	ws_kpi_35: Kpi;
	ws_kpi_36: Kpi;
	plc_inputs: classPLC32m2StatusInputs;
	plc_outputs: classPLC32m2StatusOutputs;
	ws_single_mode: Single;
	ws_cycle_mode: cycle;
	ws_cascade_mode: cascade;
	ws_mode_selector: Cascade_Cycle_Selector;
	ws_start_id_1: BOOL;
	ws_start_id_2: BOOL;
	PLC_110_32_outputs: get_status_outputs;
	out_set_frequency: classParamsValueScaling;
	hw_mode_error: WORD;
	hw_alarm_manager: ALARM_MANAGER;
	(*hw_alarm_on: BOOL;
	ws_alarm_on: BOOL;*)
	ws_mode_error: WORD;
       hw_alarm_message AT %QW8.51.0: STRING(79);
       ws_alarm_message AT %QW8.91.0: STRING(79);

	hw_external_alarm: external_alarm_invertor_drive;
	ws_external_alarm: external_alarm_invertor_drive;
END_VAR

VAR RETAIN
	hw_settings_pressure_input: SetCurrentSensorPressure_4_20;
	hw_settings_pressure_output: SetCurrentSensorPressure_4_20;
	ws_settings_pressure_input: SetCurrentSensorPressure_4_20;
	ws_settings_pressure_output: SetCurrentSensorPressure_4_20;
END_VAR
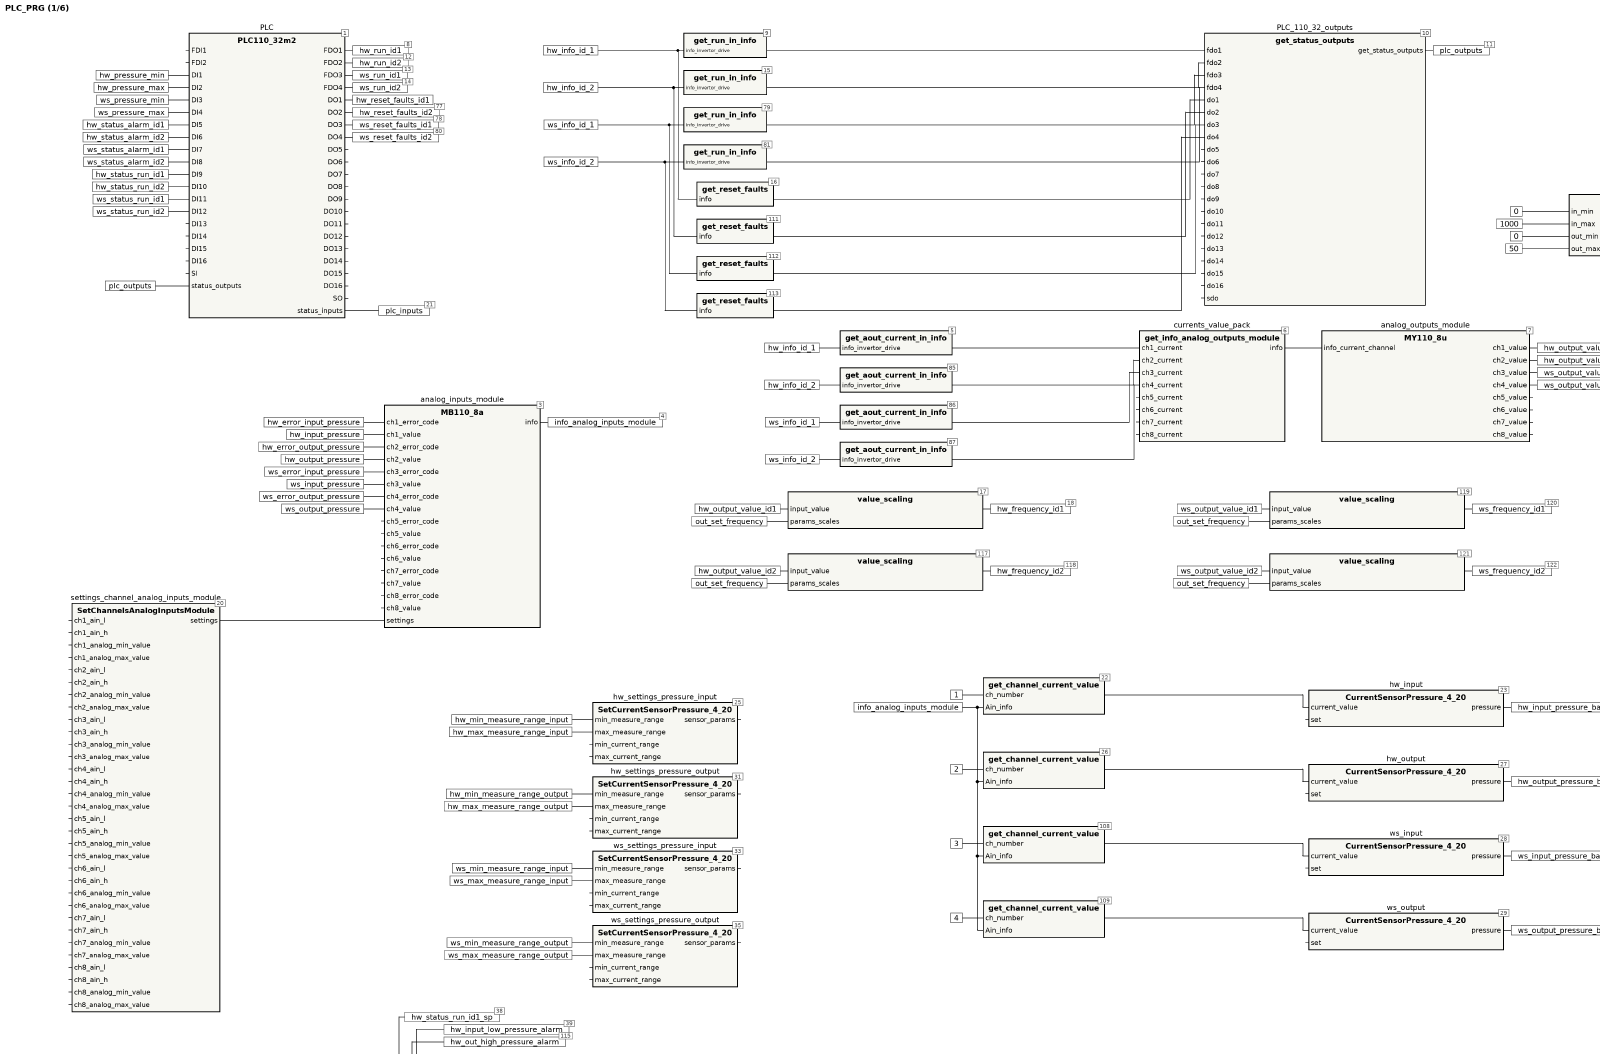
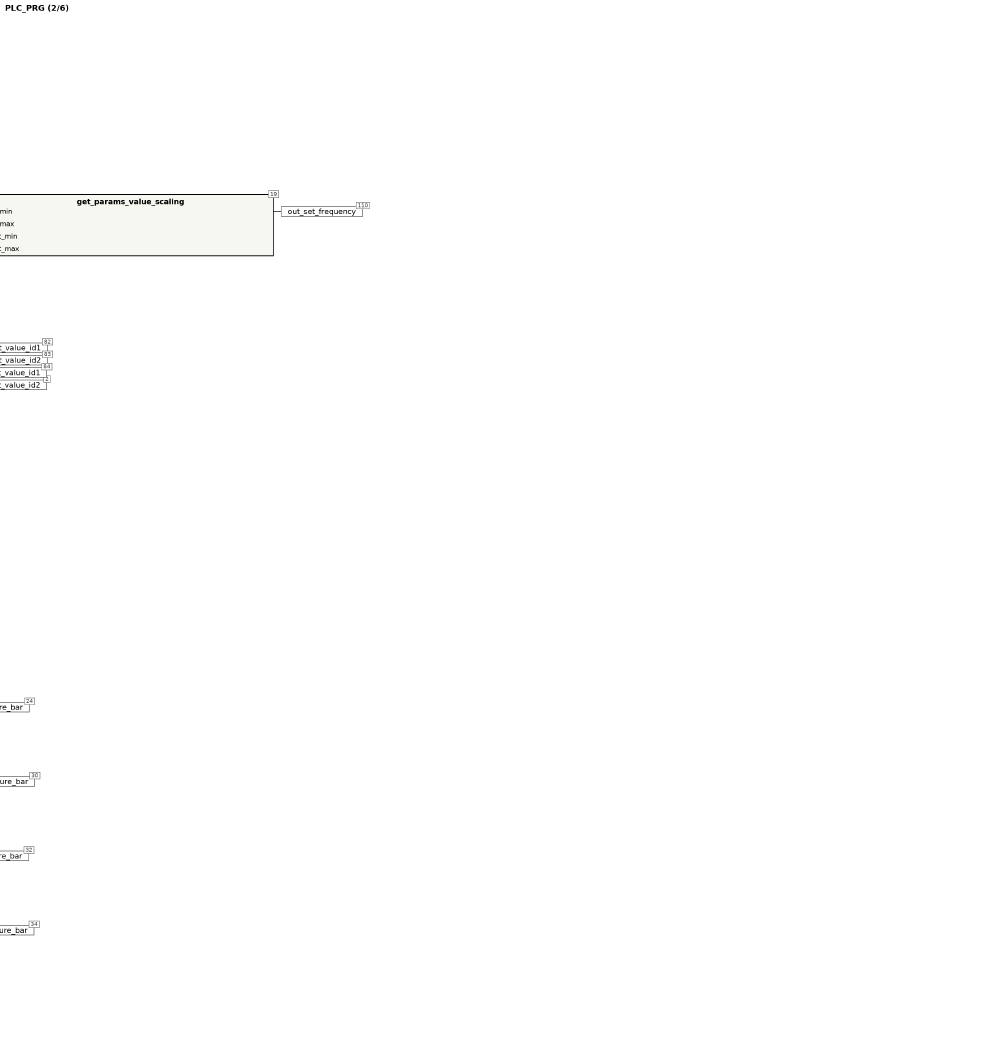
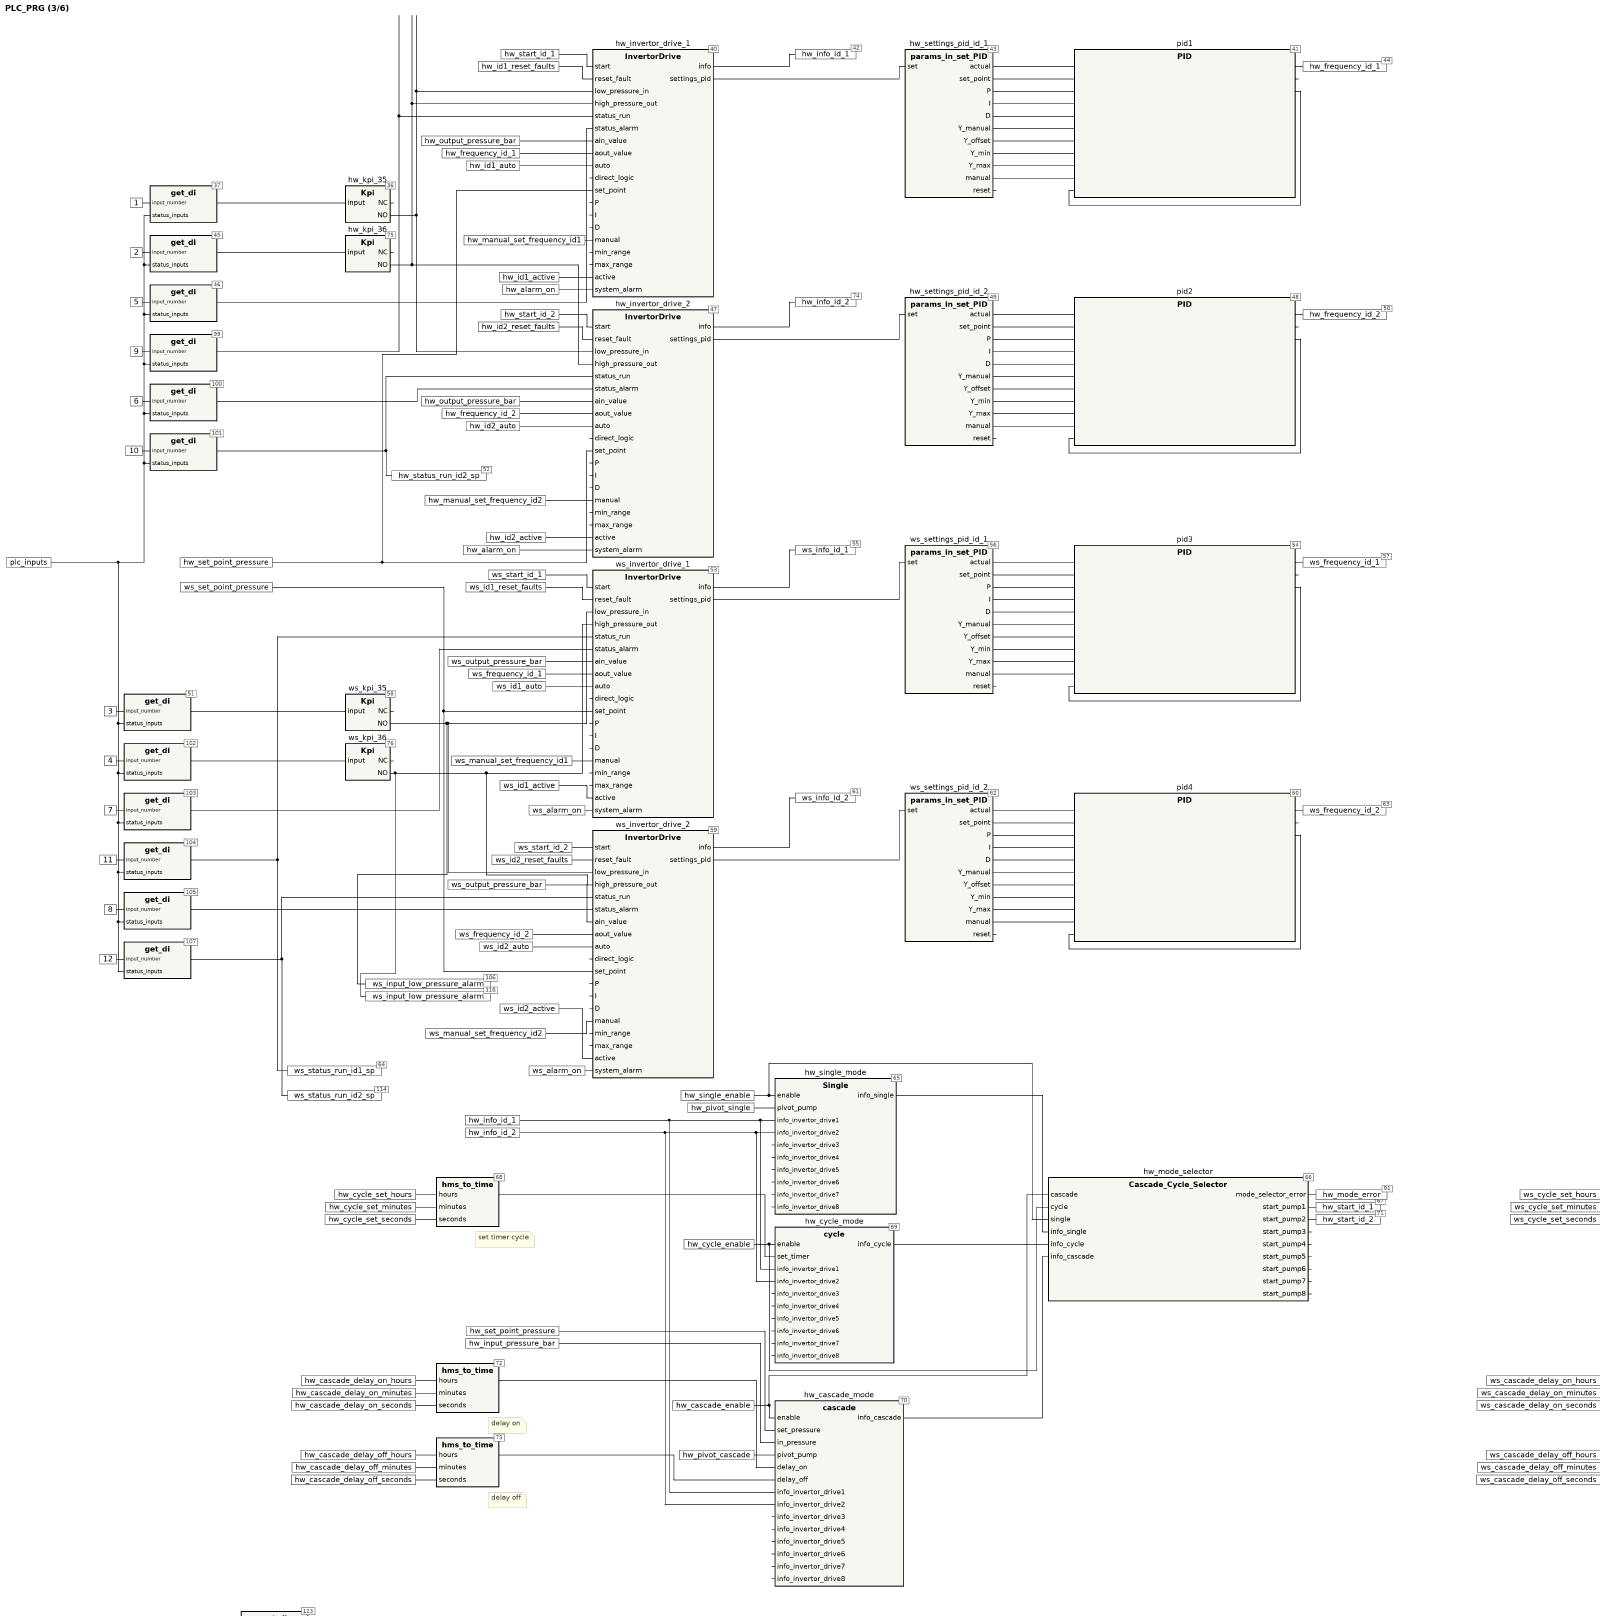
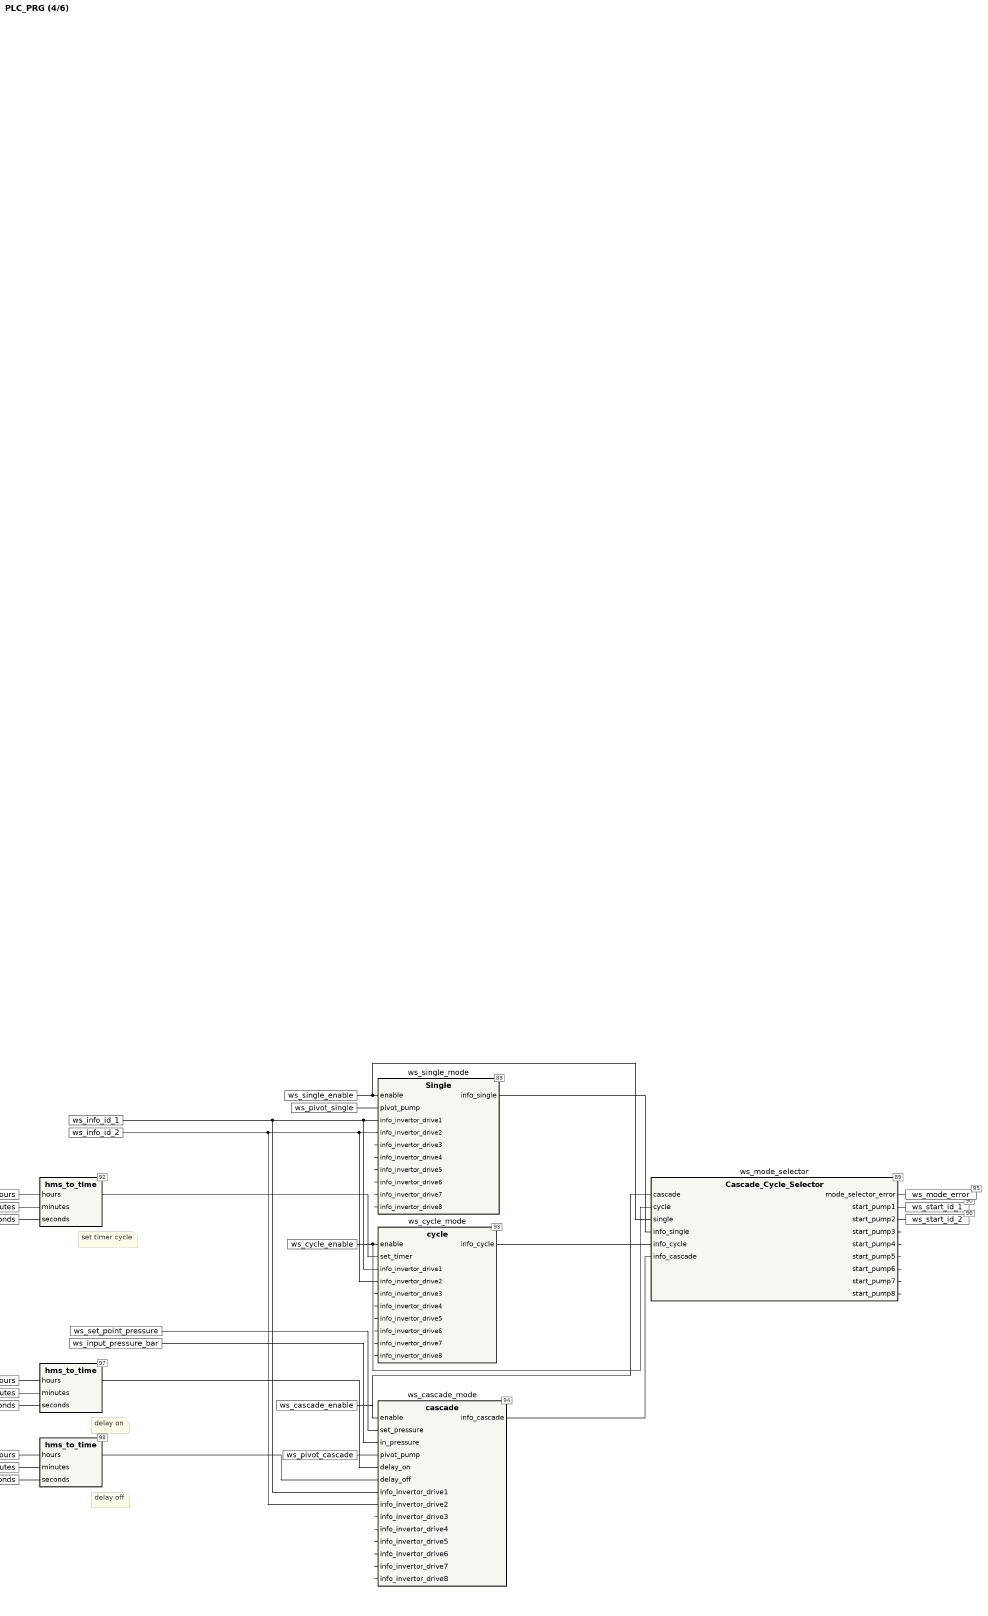
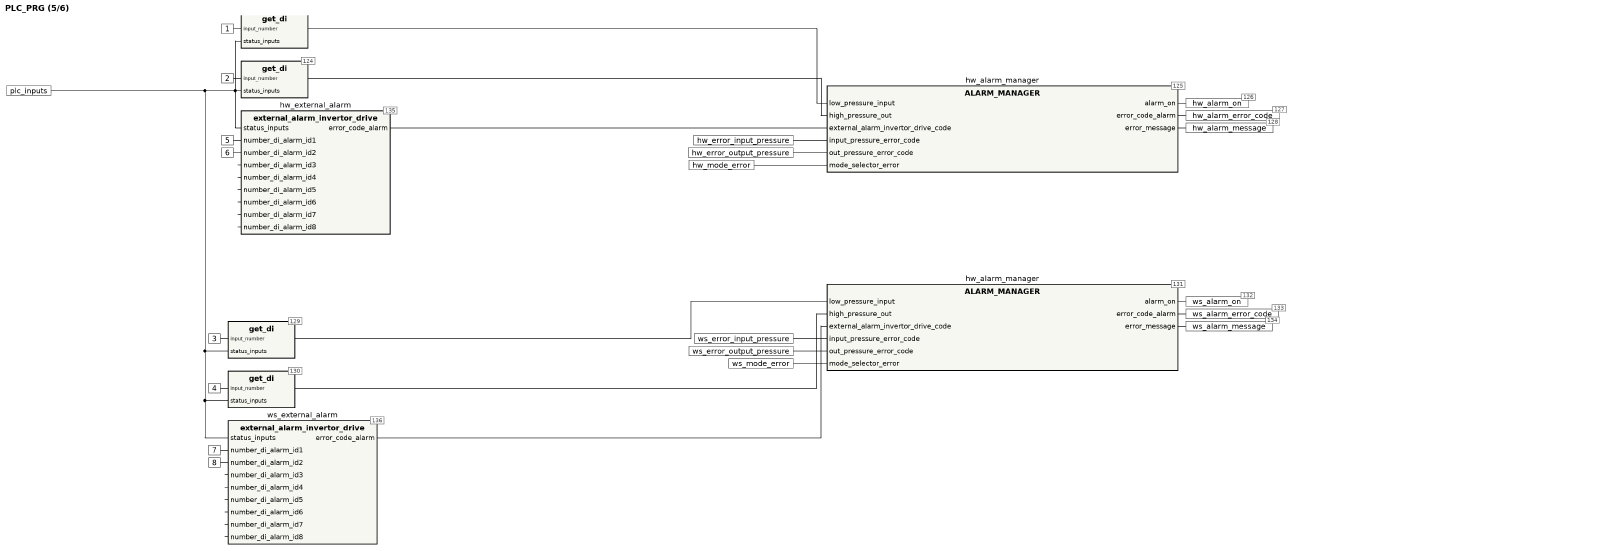
